// TIA Portal V20 export
VAR_GLOBAL   // PLC tag table "Constantes de JDT02"
   Reintentos_JDT2 AT %MB9 : USInt;
END_VAR
VAR_GLOBAL CONSTANT   // user constants
   JDT2_FinalBucleMaquinas : UInt := 500;   // Ultima Maquina del JDT02
   JDT2_FinalBucleMesas : UInt := 500;   // Ultima Mesa del JDT02
   JDT2_IdentEmisor : DInt := 'PLC1';   // Identificador del Emisor MFS (JdT)
   JDT2_IdentReceptor : DInt := 'JDT2';   // Identificador del Receptor PLC
   JDT2_InicioBucleMaquinas : UInt := 1;   // Primera Maquina del JDT02
   JDT2_InicioBucleMesas : UInt := 1;   // Primera Mesa del JDT02
   JDT2_MaxBytes : UInt := 6000;   // Maximos numeros de Bytes para enviar o recibir por TCP (8192 Bytes)
   JDT2_NDB_AKEmi : UInt := 706;   // Numero de de la Emision AK
   JDT2_NDB_EmiMensaje : UInt := 703;   // Numero de DB de la Emisión del Mensaje hacia el MFS (JdT)
   JDT2_NDB_EventosEmi : UInt := 707;   // Numero de DB de la Lista de Eventos Generados
   JDT2_NDB_EventosRec : UInt := 708;   // Numero de DB de la Lista de Eventos Recibidos
   JDT2_NDB_RecMensaje : UInt := 702;   // Numero de DB de la Recepción del Mensaje del MFS (JdT)
   JDT2_NDB_UltimoEmi : UInt := 705;   // Numero de DB del Ultimo Mensaje Enviado
   JDT2_NDB_UltimoRec : UInt := 704;   // Numero de DB del Ultimo Mensaje Recibido
   JDT2_TMPEnvioKA : UInt := 60;   // Tiempo de Espera para el Envio del Keep-Alive - 1 Minuto
   JDT2_TMPEsperaAK : UInt := 10;   // Tiempo de Espera para recibir la Confirmacion del Mensaje Enviado - 10 Segundos
   JDT2_TMPEsperaKA : UInt := 120;   // Tiempo Maximo de Espera para recibir el Keep-Alive - 2 Minutos
END_VAR
